{attribute 'GeneratedUsingTerminal: EL4001-0000-0016'}
{attribute addProperty BoxType "EL4001-0000-0016"}
{attribute addProperty Id "AO_OutputsAT %Q*AO_Outputs_BA7EBB7C2WcStateAT %I*WcState_0B2B16F91InfoDataAT %I*InfoData_32EB74EA10"}
{attribute addProperty CRC "2685036672"}
{attribute addProperty Size "13"}
TYPE EL4001_A00A6880 :
STRUCT
	{attribute addProperty Name "AO_Outputs"}
	AO_Outputs : AO_Outputs_BA7EBB7C;
	{attribute addProperty Name "WcState"}
	WcState : WcState_0B2B16F9;
	{attribute addProperty Name "InfoData"}
	InfoData : InfoData_32EB74EA;
END_STRUCT
END_TYPE

(* stored: Version 1.2.0.0, ProductVersion 3.1.4024.9
   DUT EL4001_A00A6880: Id {f5a67943-c8f5-41da-8a17-0d1ba93e29f8} *)
